// TIA Portal V15.1 export
// export: Created 2022-09-27T21:37:31.4999297Z, ExportSetting WithDefaults, WithReadOnly, DisplayName Totally Integrated Automation Portal, DisplayVersion V15.1 Update 5, DisplayName TIA Portal Openness, DisplayVersion V15.1 Update 5, DisplayName STEP 7 Professional, DisplayVersion V15.1 Update 5, DisplayName WinCC Advanced, DisplayVersion V15.1 Update 5
FUNCTION "Block_1" : Void   // FC1, LAD
{ S7_Optimized_Access := 'TRUE' }
VERSION : 0.1
// stored: AutoNumber true, CodeModifiedDate 2022-09-27T21:36:53.2302074Z, CompileDate 2022-09-27T21:36:54.6762053Z, CreationDate 2022-09-27T21:31:43.3127727Z, HandleErrorsWithinBlock false, InterfaceModifiedDate 2022-09-27T21:32:29.2295254Z, IsConsistent true, IsIECCheckEnabled false, IsKnowHowProtected false, IsWriteProtected false, LibraryConformanceStatus The object is library-conformant., ModifiedDate 2022-09-27T21:36:53.2302074Z, ParameterModified 2022-09-27T21:32:29.2295254Z, PLCSimAdvancedSupport true, SetENOAutomatically False, StructureModified 2022-09-27T21:32:29.2295254Z, UDAEnableTagReadback false
   VAR_INPUT
      Tag1 : Bool;
      Tag2 : Bool;
      Tag3 : Bool;
      Tag4 : Bool;
   END_VAR
   VAR_OUTPUT
      Tag5 : Bool;
      Tag6 : Bool;
   END_VAR
   VAR_TEMP   // added for the SCL form of the ladder/FBD networks
      _w1 : Bool;
   END_VAR
BEGIN

REGION Network 1
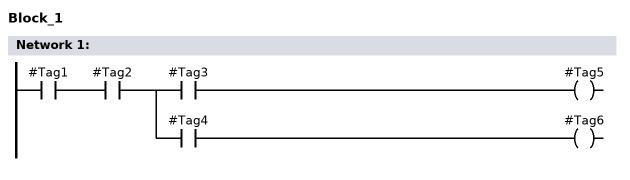
   RUNG wire#powerrail
      Contact( #Tag1 )
      Contact( #Tag2 )
      wire#w1
      Contact( #Tag3 )
      Coil( #Tag5 )
   END_RUNG
   RUNG wire#w1
      Contact( #Tag4 )
      Coil( #Tag6 )
   END_RUNG
   // the same network as SCL:
   #_w1 := #Tag1 AND #Tag2;
   #Tag5 := #_w1 AND #Tag3;
   #Tag6 := #_w1 AND #Tag4;
END_REGION
END_FUNCTION
